// TIA Portal V19 export
TYPE "CoilHandling_Persistent"
   STRUCT
      Data : Struct
         MaterialPresence : Bool;
         MaterialPresence_Decoiler : Bool;
         MaterialPresence_StraightenerEntry : Bool;
         MaterialPresence_StraightenerExit : Bool;
         MaterialPresence_JBPinchExit : Bool;
         MaterialPresence_RF_Entry : Bool;
         MaterialFullLoaded : Bool;
         VelocityOverride : Real;
         MATERIAL_SEPARATION : Struct
            Mem : Bool;
            CutDoneAndConfirmed : Bool;
         END_STRUCT;
         END_OF_COIL : Struct
            Mem : Bool;
            Tail_ReachCutPosition : Bool;
            Tail_CutDone : Bool;
            Tail_ReachJunctionPos : Bool;
            SaveEncPosAx_EndOfMaterialStraightEntry : LReal;
            SaveEncPosAx_EndOfMaterialStraightExit : LReal;
            SaveEncPosMat_CutDone : LReal;
         END_STRUCT;
         CoilLoadedInDecoiler1 : Bool;
         CoilLoadedInDecoiler2 : Bool;
         Thickness : "Thickness_PersData";
      END_STRUCT;
      Par : Struct
         MaterialBkw_PercentageStraightener : Real;
         ExtraLowSpeed_Percentage : Real;
         TimeStopInactivity : Time;
         SemiAut : Struct
            Vel_Fwd : Real;
            Vel_Bkw : Real;
            Acc : Real;
            Dec : Real;
            Jerk : Real;
         END_STRUCT;
         CoilEnd : Struct
            EnableCoilTailSequence : Bool;
            Distance_StraightEntry_To_StraightExit : LReal;   // NON USATO SU QUESTA MACCHINA
            Distance_StraightEntry_To_CutExecution : LReal;   // NON USATO SU QUESTA MACCHINA
            Distance_StraightEntry_to_JunctionExecution : LReal;   // NON USATO SU QUESTA MACCHINA
            Distance_CutHead_to_JB : LReal;
            Tol_CheckSensorStraightExit : LReal;   // NON USATO SU QUESTA MACCHINA
            Tol_PosCutExecution : LReal;   // NON USATO SU QUESTA MACCHINA
            Tol_PosJunctionExecution : LReal;   // NON USATO SU QUESTA MACCHINA
            Delay_PinchrollFwd : Time;
            Delay_StraightnerBwd : Time;
            Delay_StraightnerFwd : Time;
            Vel : LReal;
            Acc : LReal;
            Dec : LReal;
            Jerk : LReal;
            PercentageStraightener : LReal;   // % Reduction when feed with JB Pinch-roll
         END_STRUCT;
         Thickness : "Thickness_Par";
      END_STRUCT;
   END_STRUCT;
END_TYPE
